FUNCTION_BLOCK FB_FillLevel
VAR_INPUT
	nLevelIn : UINT;
	nMaxLevel : REAL;
END_VAR
VAR_OUTPUT
	nLevelPercent : REAL := 0;
	nLevelGramm : REAL := 0;
END_VAR
VAR
END_VAR

nLevelPercent := F_map(nLevelIn, 0, 32767, 100, 0);
nLevelGramm := F_map(nLevelIn, 0, 32767, nMaxLevel, 0);

END_FUNCTION_BLOCK

(* stored: Version 1.1.0.1, ProductVersion 3.1.4024.6
   POU FB_FillLevel: Id {9a1a4155-e048-4d31-8a5e-fba185ab5b97}, SpecialFunc None *)
